// LS Electric XG5000 project: 8_22
// PLC LSPLC

PROGRAM NewProgram (task: 스캔 프로그램)

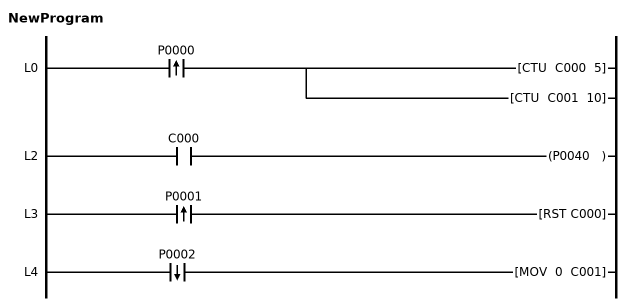
; L0
LOADP     P0000
CTU       C000 5
CTU       C001 10
; L2
LOAD      C000
OUT       P0040
; L3
LOADP     P0001
RST       C000
; L4
LOADN     P0002
MOV       0 C001